% RSLogix 500 project INTRO TO PLC - JOB 05.RSS, saved by version 10.00.00.00 %
PROJECT "PL06B"    % processor: Bul.1763 MicroLogix 1100 Series B %

PROGRAM FILES
  LAD 2   3 rungs

DATA FILES
  O0 OUTPUT  4 elements
  I1 INPUT  6 elements
  S2 STATUS  66 elements
  B3 BINARY  1 elements
  T4 TIMER  10 elements
  C5 COUNTER  2 elements
  R6 CONTROL  1 elements
  N7 INTEGER  5 elements
  F8 FLOAT  1 elements

LADDER 2
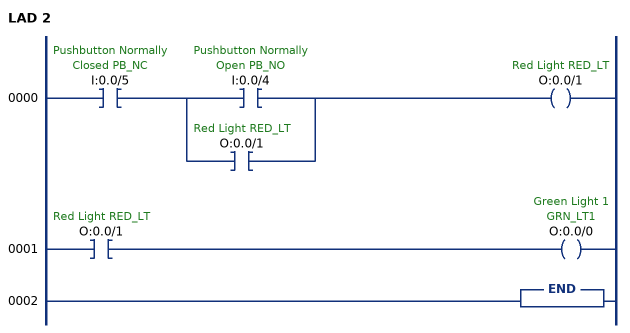
% Rung: 0 %
SOR XIC I:0.0/5 BST XIC I:0.0/4 NXB XIC O:0.0/1 BND OTE O:0.0/1 EOR
%   I:0.0/5  PB_NC  "Pushbutton Normally Closed" %
%   I:0.0/4  PB_NO  "Pushbutton Normally Open" %
%   O:0.0/1  RED_LT  "Red Light" %
% Rung: 1 %
SOR XIC O:0.0/1 OTE O:0.0/0 EOR
%   O:0.0/1  RED_LT  "Red Light" %
%   O:0.0/0  GRN_LT1  "Green Light 1" %
% Rung: 2 %
SOR END EOR

OTHER DOCUMENTED ADDRESSES
  B3:0/0  SEAL1  "Seal 1"
  B3:0/1  GRN_STOP2  "Green 2 Light Stop"
  B3:0/2  YLW_STOP  "Yellow Light Stop"
  B3:0/3  RED_STOP  "Red Light Stop"
  B3:0/4  GRN_STOP  "Green Light 1 Stop"
  B3:0/15  SCRATCH  "Scratch Bit"
  B3:1/1  RED_TMR_DNS  "Red Light Timer Done Storage"
  C5:0  HR_CTR  "Hours"
  C5:1  HOUR_CTR  "Cycle Counter 2"
  I:0.0/0  SS1A  "Selector Switch 1 Position A"
  I:0.0/1  SS1B  "Selector Switch 1 Position B"
  I:0.0/2  SS2A  "Selector Switch 2 Position A"
  I:0.0/3  SS2B  "Selector Switch 2 Position B"
  O:0.0/2  YLW_LT  "Yellow Light"
  O:0.0/3  GRN_LT2  "Green Light 2"
  RTC:0.YR  RTC
  SEL1B  
  T4:0  INT_TMR  "Light Timer"
  T4:1  YLW_TMR  "Yellow Light Timer"
  T4:2  GRN_TMR  "Green Light Timer"
  T4:3  RST_TMR  "Reset Timer"

COMMENTS NOT ATTACHED TO A CURRENT RUNG
  B3:0/0: Typical Stop Start Logic

DATA TABLE (non-zero values as saved)
DATA B3
% B3:0 % 0X800A
DATA T4
% .PRE .ACC %
% T4:0 % 40 0
% T4:1 % 5 0
% T4:2 % 5 0
% T4:3 % 10 0
DATA C5
% .PRE .ACC %
% C5:0 % 17 0
% C5:1 % 16 0
